{attribute 'GeneratedUsingTerminal: EK1100-0000-0018'}
{attribute addProperty BoxType "EK1100-0000-0018"}
{attribute addProperty Id "Beckhoff_EP6xxxEK1122Beckhoff_EP6xxxEK1122_67CC26DB1410"}
{attribute addProperty CRC "162848726"}
{attribute addProperty Size "1410"}
{attribute addProperty Name "Beckhoff EP6xxx"}
TYPE Beckhoff_EP6xxx_09B4DFD6 EXTENDS EK1100_1FC0878B :
STRUCT
	{attribute addProperty Name "Beckhoff EP6xxxEK1122"}
	{attribute addProperty PreviousPort "Beckhoff EP6xxx : B"}
	Beckhoff_EP6xxxEK1122 : Beckhoff_EP6xxxEK1122_67CC26DB;
END_STRUCT
END_TYPE

(* stored: Version 1.2.0.0, ProductVersion 3.1.4024.11
   DUT Beckhoff_EP6xxx_09B4DFD6: Id {b2d33965-7609-4b59-8053-002d0c038b0b} *)
